// TIA Portal project "proyecto final" (V14)

(* hardware
DEVICE "S7-1200 station_1"  S7-1200 Station
   slot 0: "Rack_0"  S7-1200 Rack  Rack  V1.0
   slot 1: "PLC_1"  CPU 1214C AC/DC/Rly  6ES7 214-1BG40-0XB0  V4.1
*)

// ===== PLC "PLC_1"  CPU 1214C AC/DC/Rly =====

VAR_GLOBAL   // PLC tag table "Tabla de variables estándar"
   "on" AT %M2.0 : Bool;
   "Tag_1" AT %M2.1 : Bool;
   "planta" AT %Q0.0 : Bool;
   "Tag_2" AT %MD34 : DWord;
   "Tag_3" AT %IW66 : Word;
   "Tag_4" AT %IW64 : Word;
   "voltaje" AT %MD20 : Real;
   "bomba" AT %Q0.1 : Bool;
   "apagar bomba" AT %M3.4 : Bool;
   "Tag_5" AT %MD30 : Real;
   "Tag_6" AT %MD50 : Real;
   "Histeresis" AT %MD6 : Real;
   "Nivel Maximo" AT %MD600 : Real;
   "Tag_7" AT %M1000.0 : Bool;
   "Tag_8" AT %M1000.1 : Bool;
   "Tag_9" AT %M1000.3 : Bool;
   "Tag_10" AT %M102.0 : Bool;
   "Tag_11" AT %I0.0 : Bool;
   "Tag_12" AT %I0.1 : Bool;
   "Tag_13" AT %M19.7 : Bool;
   "Tag_14" AT %M20.0 : Bool;
   "Tag_15" AT %M2005.0 : Bool;
END_VAR

ORGANIZATION_BLOCK "Main"   // OB1, LAD, ProgramCycle
TITLE = "Main Program Sweep (Cycle)"
{ S7_Optimized_Access := 'TRUE' }
VERSION : 0.1
   VAR_INPUT
      Initial_Call : Bool;   // Initial call of this OB
      Remanence : Bool;   // =True, if remanent data are available
   END_VAR
BEGIN

REGION Network 1
   // control on/off de la planta
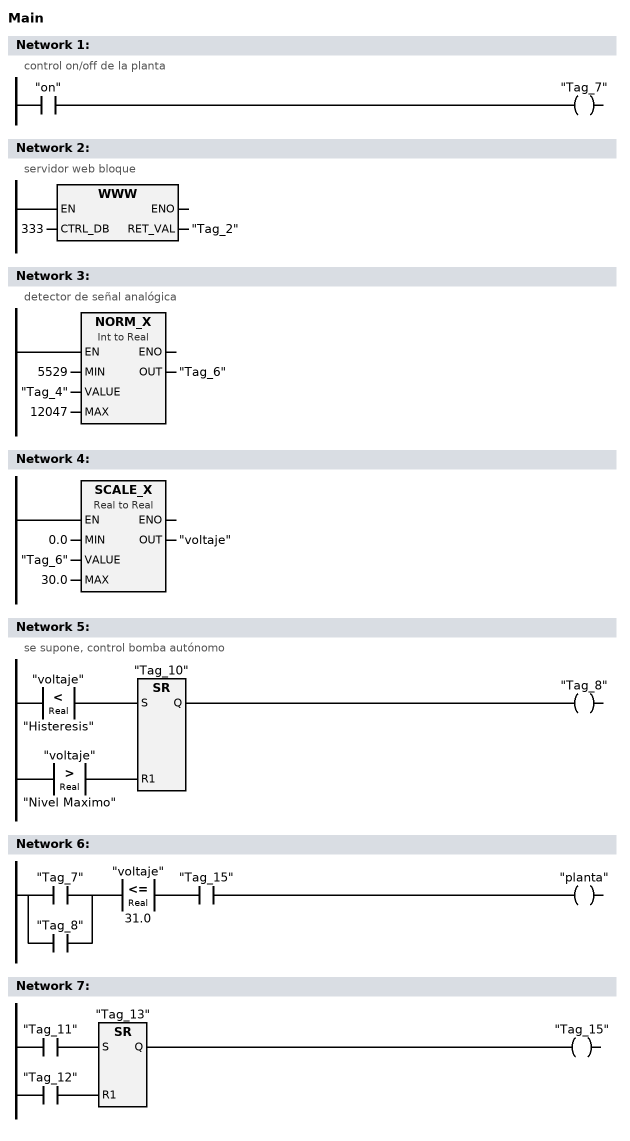
   RUNG wire#powerrail
      Contact( "on" )
      Coil( "Tag_7" )
   END_RUNG
   // the same network as SCL:
   "Tag_7" := "on";
END_REGION

REGION Network 2
   // servidor web bloque
   "Tag_2" := WWW(CTRL_DB := 333);
END_REGION

REGION Network 3
   // detector de señal analógica
   RUNG wire#powerrail
      { S7_Templates := "[SrcType := Int, DestType := Real]" } Normalize(min := 5529, value := "Tag_4", max := 12047, out => "Tag_6")
   END_RUNG
   // the same network as SCL:
   "Tag_6" := NORM_X(MIN := 5529, VALUE := "Tag_4", MAX := 12047);
END_REGION

REGION Network 4
   RUNG wire#powerrail
      { S7_Templates := "[SrcType := Real, DestType := Real]" } Scale(min := 0.0, value := "Tag_6", max := 30.0, out => "voltaje")
   END_RUNG
   // the same network as SCL:
   "voltaje" := SCALE_X(MIN := 0.0, VALUE := "Tag_6", MAX := 30.0);
END_REGION

REGION Network 5
   // se supone, control bomba autónomo
   RUNG wire#powerrail
      { S7_Templates := "SrcType := Real" } LT_Contact(in1 := "voltaje", in2 := "Histeresis")
      S_SR(operand := "Tag_10", r1 := wire#w1)
      Coil( "Tag_8" )
   END_RUNG
   RUNG wire#powerrail
      { S7_Templates := "SrcType := Real" } GT_Contact(in1 := "voltaje", in2 := "Nivel Maximo")
   END_RUNG wire#w1
   // the same network as SCL:
   IF "voltaje" < "Histeresis" THEN
       "Tag_10" := TRUE;   // SR flip-flop
   END_IF;
   IF "voltaje" > "Nivel Maximo" THEN "Tag_10" := FALSE; END_IF;
   "Tag_8" := "Tag_10";
END_REGION

REGION Network 6
   RUNG wire#powerrail
      Contact( "Tag_7" )
      wire#w1
      { S7_Templates := "SrcType := Real" } LE_Contact(in1 := "voltaje", in2 := 31.0)
      Contact( "Tag_15" )
      Coil( "planta" )
   END_RUNG
   RUNG wire#powerrail
      Contact( "Tag_8" )
   END_RUNG wire#w1
   // the same network as SCL:
   "planta" := ("Tag_7" OR "Tag_8") AND ("voltaje" <= 31.0) AND "Tag_15";
END_REGION

REGION Network 7
   RUNG wire#powerrail
      Contact( "Tag_11" )
      S_SR(operand := "Tag_13", r1 := wire#w1)
      Coil( "Tag_15" )
   END_RUNG
   RUNG wire#powerrail
      Contact( "Tag_12" )
   END_RUNG wire#w1
   // the same network as SCL:
   IF "Tag_11" THEN
       "Tag_13" := TRUE;   // SR flip-flop
   END_IF;
   IF "Tag_12" THEN "Tag_13" := FALSE; END_IF;
   "Tag_15" := "Tag_13";
END_REGION
END_ORGANIZATION_BLOCK